PROGRAM Camera
VAR
		cameraData : CameraConnectionUDP;
		soc : SoC_Calc;
END_VAR

cameraData();
soc();
Main.setIstPoseCamera(PoseArray := cameraData.robotPosition);

METHOD getX : LREAL
VAR_INPUT
	robot_number : int;
END_VAR
//return cameraData.robotposition[robot_number].x;
END_METHOD

END_PROGRAM

(* stored: Version 1.1.0.1, ProductVersion 3.1.4024.11
   POU Camera: Id {f47d8b4d-3b12-40ce-95f8-97ff406a7170}, SpecialFunc None
   Method getX: Id {14032c57-2b4d-42cb-8fce-631bf67d0508} *)
